(* PLC project Rasi_feeds_batching.project, Automation Builder 2.7 - Basic Automation Builder 2.7 *)
(* stored: creationDateTime 2026-08-27T17:40:00 *)

PROGRAM batching14
  VAR
    Supervisor_Inst : Batch_Supervisor_V14;
    Auto_Ctrl_Inst : Auto_Batching_V14;
    Semi_Auto_Ctrl_Inst : Semi_Auto_Batching_V14;
    Auto_Complete : BOOL;
    Semi_Auto_Complete : BOOL;
    Auto_Err : INT;
    Auto_Msg : STRING;
    Semi_Auto_Err : INT;
    Semi_Auto_Msg : STRING;
  END_VAR

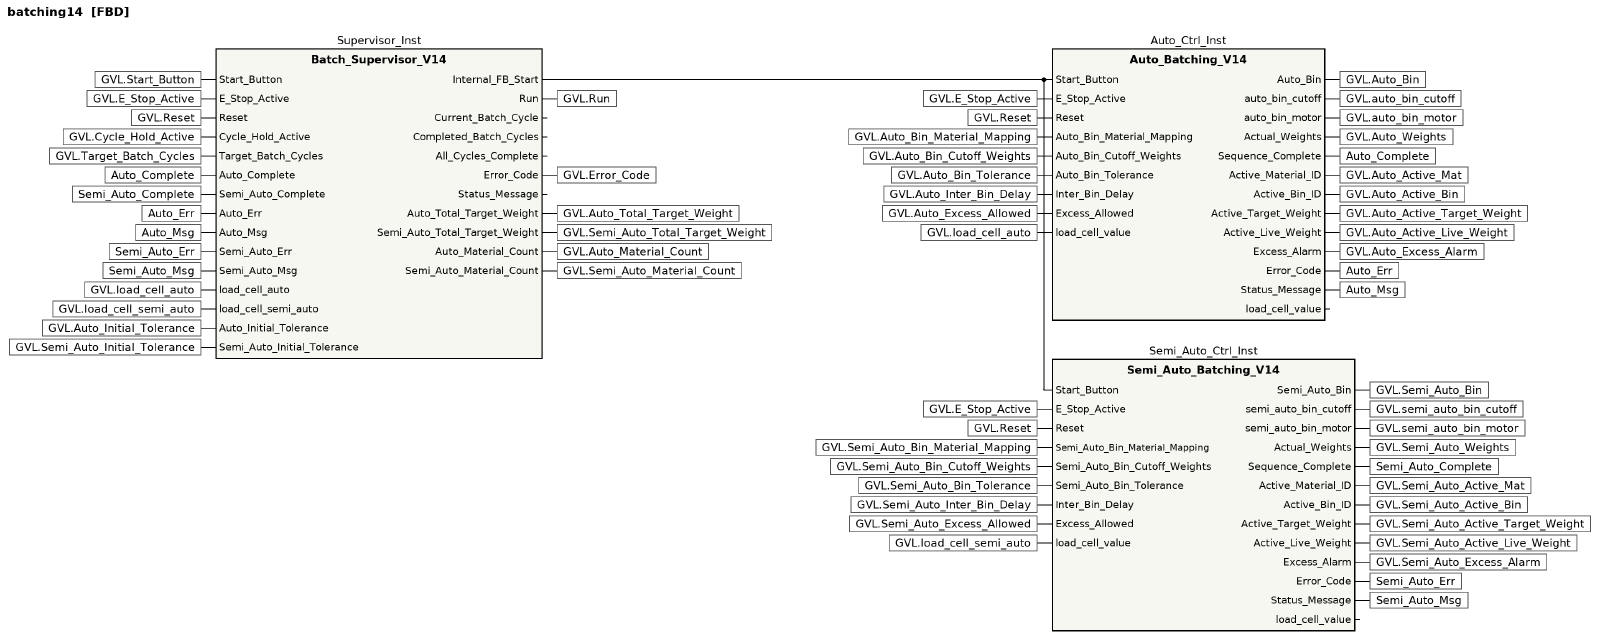
(* FBD diagram, written out as Structured Text *)
Supervisor_Inst(Start_Button := GVL.Start_Button, E_Stop_Active := GVL.E_Stop_Active, Reset := GVL.Reset, Cycle_Hold_Active := GVL.Cycle_Hold_Active, Target_Batch_Cycles := GVL.Target_Batch_Cycles, Auto_Complete := Auto_Complete, Semi_Auto_Complete := Semi_Auto_Complete, Auto_Err := Auto_Err, Auto_Msg := Auto_Msg, Semi_Auto_Err := Semi_Auto_Err, Semi_Auto_Msg := Semi_Auto_Msg, load_cell_auto := GVL.load_cell_auto, load_cell_semi_auto := GVL.load_cell_semi_auto, Auto_Initial_Tolerance := GVL.Auto_Initial_Tolerance, Semi_Auto_Initial_Tolerance := GVL.Semi_Auto_Initial_Tolerance);
Auto_Ctrl_Inst(Start_Button := Supervisor_Inst.Internal_FB_Start, E_Stop_Active := GVL.E_Stop_Active, Reset := GVL.Reset, Auto_Bin_Material_Mapping := GVL.Auto_Bin_Material_Mapping, Auto_Bin_Cutoff_Weights := GVL.Auto_Bin_Cutoff_Weights, Auto_Bin_Tolerance := GVL.Auto_Bin_Tolerance, Inter_Bin_Delay := GVL.Auto_Inter_Bin_Delay, Excess_Allowed := GVL.Auto_Excess_Allowed, load_cell_value := GVL.load_cell_auto);
Semi_Auto_Ctrl_Inst(Start_Button := Supervisor_Inst.Internal_FB_Start, E_Stop_Active := GVL.E_Stop_Active, Reset := GVL.Reset, Semi_Auto_Bin_Material_Mapping := GVL.Semi_Auto_Bin_Material_Mapping, Semi_Auto_Bin_Cutoff_Weights := GVL.Semi_Auto_Bin_Cutoff_Weights, Semi_Auto_Bin_Tolerance := GVL.Semi_Auto_Bin_Tolerance, Inter_Bin_Delay := GVL.Semi_Auto_Inter_Bin_Delay, Excess_Allowed := GVL.Semi_Auto_Excess_Allowed, load_cell_value := GVL.load_cell_semi_auto);
GVL.Run := Supervisor_Inst.Run;
GVL.Error_Code := Supervisor_Inst.Error_Code;
GVL.Auto_Total_Target_Weight := Supervisor_Inst.Auto_Total_Target_Weight;
GVL.Semi_Auto_Total_Target_Weight := Supervisor_Inst.Semi_Auto_Total_Target_Weight;
GVL.Auto_Material_Count := Supervisor_Inst.Auto_Material_Count;
GVL.Semi_Auto_Material_Count := Supervisor_Inst.Semi_Auto_Material_Count;
GVL.Auto_Bin := Auto_Ctrl_Inst.Auto_Bin;
GVL.auto_bin_cutoff := Auto_Ctrl_Inst.auto_bin_cutoff;
GVL.auto_bin_motor := Auto_Ctrl_Inst.auto_bin_motor;
GVL.Auto_Weights := Auto_Ctrl_Inst.Actual_Weights;
Auto_Complete := Auto_Ctrl_Inst.Sequence_Complete;
GVL.Auto_Active_Mat := Auto_Ctrl_Inst.Active_Material_ID;
GVL.Auto_Active_Bin := Auto_Ctrl_Inst.Active_Bin_ID;
GVL.Auto_Active_Target_Weight := Auto_Ctrl_Inst.Active_Target_Weight;
GVL.Auto_Active_Live_Weight := Auto_Ctrl_Inst.Active_Live_Weight;
GVL.Auto_Excess_Alarm := Auto_Ctrl_Inst.Excess_Alarm;
Auto_Err := Auto_Ctrl_Inst.Error_Code;
Auto_Msg := Auto_Ctrl_Inst.Status_Message;
GVL.Semi_Auto_Bin := Semi_Auto_Ctrl_Inst.Semi_Auto_Bin;
GVL.semi_auto_bin_cutoff := Semi_Auto_Ctrl_Inst.semi_auto_bin_cutoff;
GVL.semi_auto_bin_motor := Semi_Auto_Ctrl_Inst.semi_auto_bin_motor;
GVL.Semi_Auto_Weights := Semi_Auto_Ctrl_Inst.Actual_Weights;
Semi_Auto_Complete := Semi_Auto_Ctrl_Inst.Sequence_Complete;
GVL.Semi_Auto_Active_Mat := Semi_Auto_Ctrl_Inst.Active_Material_ID;
GVL.Semi_Auto_Active_Bin := Semi_Auto_Ctrl_Inst.Active_Bin_ID;
GVL.Semi_Auto_Active_Target_Weight := Semi_Auto_Ctrl_Inst.Active_Target_Weight;
GVL.Semi_Auto_Active_Live_Weight := Semi_Auto_Ctrl_Inst.Active_Live_Weight;
GVL.Semi_Auto_Excess_Alarm := Semi_Auto_Ctrl_Inst.Excess_Alarm;
Semi_Auto_Err := Semi_Auto_Ctrl_Inst.Error_Code;
Semi_Auto_Msg := Semi_Auto_Ctrl_Inst.Status_Message;
END_PROGRAM
